Universal Robots PolyScope program: Test Script Calcs.urp

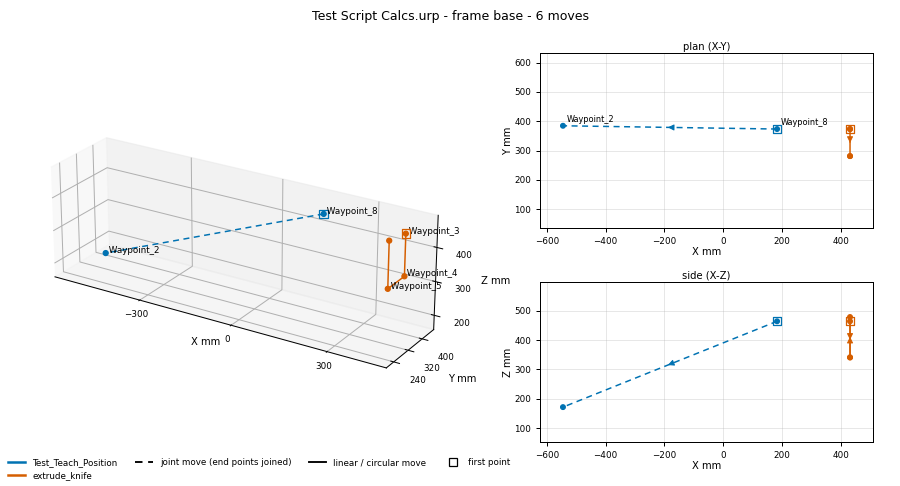
[picture p0: tool path of Test Script Calcs.urp in frame base, 6 of 9 moves have a stored position in this frame; points joined in program order, loops and branches not executed]
Program Test Script Calcs (installation=default directory=/programs createdIn=5.14.5 lastSavedIn=5.14.5 robotSerialNumber=20236801216)
Calibrated DH parameters: a=[-0.000021, -0.748897, -0.28186, -0.00004, -0.000055, 0]; d=[0.236225, -424.082933, -1564.66872, 1988.95162, 0.159094, 0.153873]; alpha=[1.570844, 0.001002, 0.000337, 1.571488, -1.569996, 0]; deltaTheta=[0, -0.516316, 5.626292, 1.173211, 0.000001, 0]
InitVariablesNode variables(variable(name=freedrive_m_var, expression=False))
Robot Program (runOnlyOnce=true)
  Script: Test_Teach_Position()
  Script: Corner_Homing_BRB()
  Script: extrude_knife()
  Script: test_script_calcs2()
SubProgram Test_Teach_Position (keepSynchronizedWithDisk=false) programFile=/programs/Test Teach Position.urp
  SafeHome (positionOptionType=SPEED_AND_ACCELERATION speed=1.047198 acceleration=1.396263 nextMotionTime=2)
  MoveL speed 250 mm/s, acceleration 1200 mm/s^2 (useActiveTCP=true) feature=Base
    Waypoint Waypoint_8: TCP in base x=183.613 y=373.491 z=464.002 mm, rx=0 ry=3.1416 rz=0 rad; joints [-144.817, -120.486, 148.461, -117.931, -90.033, 125.101] deg; TCP offset x=0 y=0 z=19 mm, rx=0 ry=0 rz=0 rad
    'move welder up out of holder'
  MoveJ speed 60 deg/s, acceleration 80 deg/s^2 (useActiveTCP=true) feature=Base
    Waypoint Waypoint_2: TCP in base x=-545.552 y=384.638 z=171.639 mm, rx=0.6685 ry=-1.9493 rz=1.7266 rad; joints [-60.534, -62.274, 125.356, -70.677, -59.999, 145.088] deg
  freedrive_m_var := False
  freedrive_m_var := True
  Popup Message (haltProgram=false message=Move the robot to the peg center, then click 'Continue' inputType=Text)
  freedrive_m_var := False
  Wait Sleep waitTime=0.25
  Script: sync()
  tcp_pose := get_actual_joint_positions()
SubProgram Corner_Homing_BRB (keepSynchronizedWithDisk=false) programFile=/programs/Corner Homing BRB.urp
  'Use this program when tool is already positioned close to corner (back right bottom corner)'
  'tool flange will seek all 3 sides and then bring tcp to the corner'
  Script: align_tcp_left()
  'right side'
  MoveL speed 250 mm/s, acceleration 1200 mm/s^2 (useActiveTCP=true) feature=Base
    MoveDirectionNode (selectedDirection=XMinus)
      Until DISTANCE (allowActions=false deceleration=3 distanceNodeType=STOP) Distance=0.05; motionParameters(blendRadius=0)
  MoveL speed 50 mm/s, acceleration 1200 mm/s^2 (useActiveTCP=true) feature=Base
    MoveDirectionNode (selectedDirection=YMinus)
      Until TOOL_CONTACT_DETECTION (allowActions=false retraction=0 decelerationAcceleration=3 decelerationAngularAcceleration=34.906585)
  p11 := get_actual_tcp_pose()
  MoveL speed 250 mm/s, acceleration 1200 mm/s^2 (useActiveTCP=true) feature=Base
    MoveDirectionNode (selectedDirection=YPlus)
      Until DISTANCE (allowActions=false deceleration=3 distanceNodeType=STOP) Distance=0.05; motionParameters(blendRadius=0)
  MoveL speed 250 mm/s, acceleration 1200 mm/s^2 (useActiveTCP=true) feature=Base
    MoveDirectionNode (selectedDirection=XMinus)
      Until DISTANCE (allowActions=false deceleration=3 distanceNodeType=STOP) Distance=0.05; motionParameters(blendRadius=0)
  MoveL speed 50 mm/s, acceleration 1200 mm/s^2 (useActiveTCP=true) feature=Base
    MoveDirectionNode (selectedDirection=YMinus)
      Until TOOL_CONTACT_DETECTION (allowActions=false retraction=0 decelerationAcceleration=3 decelerationAngularAcceleration=34.906585)
  p12 := get_actual_tcp_pose()
  MoveL speed 250 mm/s, acceleration 1200 mm/s^2 (useActiveTCP=true) feature=Base
    MoveDirectionNode (selectedDirection=YPlus)
      Until DISTANCE (allowActions=false deceleration=3 distanceNodeType=STOP) Distance=0.05; motionParameters(blendRadius=0)
  MoveL speed 250 mm/s, acceleration 1200 mm/s^2 (useActiveTCP=true) feature=Base
    MoveDirectionNode (selectedDirection=XPlus)
      Until DISTANCE (allowActions=false deceleration=3 distanceNodeType=STOP) Distance=0.2; motionParameters(blendRadius=0)
  Script: align_tcp_forward()
  'back side'
  MoveL speed 250 mm/s, acceleration 1200 mm/s^2 (useActiveTCP=true) feature=Base
    MoveDirectionNode (selectedDirection=YMinus)
      Until DISTANCE (allowActions=false deceleration=3 distanceNodeType=STOP) Distance=0.1; motionParameters(blendRadius=0)
  MoveL speed 50 mm/s, acceleration 1200 mm/s^2 (useActiveTCP=true) feature=Base
    MoveDirectionNode (selectedDirection=XMinus)
      Until TOOL_CONTACT_DETECTION (allowActions=false retraction=0 decelerationAcceleration=3 decelerationAngularAcceleration=34.906585)
  p21 := get_actual_tcp_pose()
  MoveL speed 250 mm/s, acceleration 1200 mm/s^2 (useActiveTCP=true) feature=Base
    MoveDirectionNode (selectedDirection=XPlus)
      Until DISTANCE (allowActions=false deceleration=3 distanceNodeType=STOP) Distance=0.05; motionParameters(blendRadius=0)
  MoveL speed 250 mm/s, acceleration 1200 mm/s^2 (useActiveTCP=true) feature=Base
    MoveDirectionNode (selectedDirection=YMinus)
      Until DISTANCE (allowActions=false deceleration=3 distanceNodeType=STOP) Distance=0.05; motionParameters(blendRadius=0)
  MoveL speed 50 mm/s, acceleration 1200 mm/s^2 (useActiveTCP=true) feature=Base
    MoveDirectionNode (selectedDirection=XMinus)
      Until TOOL_CONTACT_DETECTION (allowActions=false retraction=0 decelerationAcceleration=3 decelerationAngularAcceleration=34.906585)
  p22 := get_actual_tcp_pose()
  MoveL speed 250 mm/s, acceleration 1200 mm/s^2 (useActiveTCP=true) feature=Base
    MoveDirectionNode (selectedDirection=XPlus)
      Until DISTANCE (allowActions=false deceleration=3 distanceNodeType=STOP) Distance=0.05; motionParameters(blendRadius=0)
  'regroup for up turn'
  MoveL speed 250 mm/s, acceleration 1200 mm/s^2 (useActiveTCP=true) feature=Base
    MoveDirectionNode (selectedDirection=XPlus)
      Until DISTANCE (allowActions=false deceleration=3 distanceNodeType=STOP) Distance=0.2; motionParameters(blendRadius=0)
    MoveDirectionNode (selectedDirection=YPlus)
      Until DISTANCE (allowActions=false deceleration=3 distanceNodeType=STOP) Distance=0.4; motionParameters(blendRadius=0)
  MoveL speed 250 mm/s, acceleration 1200 mm/s^2 (useActiveTCP=true) feature=Base
    MoveDirectionNode (selectedDirection=ZMinus)
      Until DISTANCE (allowActions=false deceleration=3 distanceNodeType=STOP) Distance=0.1; motionParameters(blendRadius=0)
  Script: align_tcp_up()
  MoveL speed 250 mm/s, acceleration 1200 mm/s^2 (useActiveTCP=true) feature=Base
    MoveDirectionNode (selectedDirection=XMinus)
      Until DISTANCE (allowActions=false deceleration=3 distanceNodeType=STOP) Distance=0.25; motionParameters(blendRadius=0)
    MoveDirectionNode (selectedDirection=YMinus)
      Until DISTANCE (allowActions=false deceleration=3 distanceNodeType=STOP) Distance=0.3; motionParameters(blendRadius=0)
  'bottom side'
  MoveL speed 250 mm/s, acceleration 1200 mm/s^2 (useActiveTCP=true) feature=Base
    MoveDirectionNode (selectedDirection=YMinus)
      Until DISTANCE (allowActions=false deceleration=3 distanceNodeType=STOP) Distance=0.12; motionParameters(blendRadius=0)
  MoveL speed 50 mm/s, acceleration 1200 mm/s^2 (useActiveTCP=true) feature=Base
    MoveDirectionNode (selectedDirection=ZPlus)
      Until TOOL_CONTACT_DETECTION (allowActions=false retraction=0 decelerationAcceleration=3 decelerationAngularAcceleration=34.906585)
  p3 := get_actual_tcp_pose()
  MoveL speed 250 mm/s, acceleration 1200 mm/s^2 (useActiveTCP=true) feature=Base
    MoveDirectionNode (selectedDirection=ZMinus)
      Until DISTANCE (allowActions=false deceleration=3 distanceNodeType=STOP) Distance=0.05; motionParameters(blendRadius=0)
  MoveL speed 250 mm/s, acceleration 1200 mm/s^2 (useActiveTCP=true) feature=Base
    MoveDirectionNode (selectedDirection=XPlus)
      Until DISTANCE (allowActions=false deceleration=3 distanceNodeType=STOP) Distance=0.1; motionParameters(blendRadius=0)
    MoveDirectionNode (selectedDirection=YPlus)
      Until DISTANCE (allowActions=false deceleration=3 distanceNodeType=STOP) Distance=0.1; motionParameters(blendRadius=0)
SubProgram extrude_knife (keepSynchronizedWithDisk=false) programFile=/programs/extrude_knife.urp
  'Move to bucket'
  MoveJ speed 60 deg/s, acceleration 80 deg/s^2 (useActiveTCP=true) feature=Base
    Waypoint Waypoint_3: TCP in base x=432.121 y=373.496 z=463.993 mm, rx=0 ry=-3.1416 rz=0 rad; joints [-159.589, -103.956, 140.658, -126.656, -90.019, 110.321] deg
  MoveL speed 250 mm/s, acceleration 1200 mm/s^2 (useActiveTCP=true) feature=Base
    Waypoint Waypoint_4: TCP in base x=432.138 y=373.502 z=340.884 mm, rx=0 ry=3.1416 rz=0 rad; joints [-159.596, -94.144, 147.137, -142.947, -90.01, 110.313] deg
  'extrude out a foot'
  Wait Sleep waitTime=6
  MoveL speed 40 mm/s, acceleration 1200 mm/s^2 (useActiveTCP=true) feature=Base
    'slice over knife'
    Waypoint Waypoint_5: TCP in base x=432.16 y=281.352 z=340.893 mm, rx=0 ry=3.1416 rz=0 rad; joints [-169.69, -98.838, 150.801, -141.919, -90.013, 100.22] deg
  MoveL speed 250 mm/s, acceleration 1200 mm/s^2 (useActiveTCP=true) feature=Base
    Waypoint Waypoint_6: TCP in base x=432.128 y=281.346 z=478.493 mm, rx=0 ry=-3.1416 rz=0 rad; joints [-169.679, -110.118, 142.836, -122.671, -90.025, 100.232] deg
    'raise up away from knife'
SubProgram test_script_calcs2 (keepSynchronizedWithDisk=false) programFile=/programs/test_script_calcs2.urp
  point1 := get_actual_tcp_pose()
  point2 := get_actual_tcp_pose()
  point3 := get_actual_tcp_pose()
  point4 := get_actual_tcp_pose()
  Script file /programs/analyze_touchpoints.script
    | # comment get the z
    | zcoord=p3[2]
    | 
    | # get the raw points from the first line
    | l1p1x=p11[0]
    | l1p1y=p11[1]
    | l1p2x=p12[0]
    | l1p2y=p12[1]
    | 
    | # equate the first line in 2d space
    | ml1 = (l1p2y-l1p1y) / (l1p2x-l1p1x)
    | 
    | # b = y - mx
    | bl1 = l1p1y - ml1 * l1p1x
    | 
    | # get the raw points from the second line
    | l2p1x=p21[0]
    | l2p1y=p21[1]
    | l2p2x=p22[0]
    | l2p2y=p22[1]
    | 
    | # equate the second line in 2d space
    | ml2 = (l2p2y-l2p1y) / (l2p2x-l2p1x)
    | 
    | # b = y - mx
    | bl2 = l2p1y - ml2 * l2p1x
    | 
    | 
    | # find the intersection of the two lines
    | # m1x+b1 = m2x+b2
    | # m1x - m2x = b2 - b1
    | # x = (b2-b1) / (m1-m2)
    | xintersect = (bl2-bl1) / (ml1-ml2)
    | yintersect = ml1 * xintersect + bl1
    | 
    | 
    | # find locations 8 inches away from  intersect point
    | # CONST
    | welddistance = 8
    | roundoverdistance = .25
    | zup = .375
    | # inches
    | wd = welddistance * 25.4 / 1000
    | rod = roundoverdistance * 25.4 / 1000
    | zup = zup * 25.4 / 1000
    | 
    | #define a vector from the intersection to the second point on the first line
    | l1delxfull = l1p2x - xintersect
    | l1delyfull = l1p2y - yintersect
    | 
    | l1delmag = sqrt(l1delxfull*l1delxfull + l1delyfull*l1delyfull)
    | 
    | l1delxunit = l1delxfull / l1delmag
    | l1delyunit = l1delyfull / l1delmag
    | 
    | # now we have the unit vector. extend the weld distance from the intersection
    | x = xintersect + l1delxunit * wd
    | y = yintersect + l1delyunit * wd
    | z = zcoord + zup
    | 
    | point1 = p[x,y,z,1.570796,0,0] # dummy orientation for now
    | 
    | x = xintersect + l1delxunit * rod
    | y = yintersect + l1delyunit * rod
    | 
    | point2 = p[x,y,z,1.570796,0,0]
    | 
    | #define a vector from the intersection to the second point on the second line
    | l2delxfull = l2p2x - xintersect
    | l2delyfull = l2p2y - yintersect
    | 
    | l2delmag = sqrt(l2delxfull*l2delxfull + l2delyfull*l2delyfull)
    | 
    | l2delxunit = l2delxfull / l2delmag
    | l2delyunit = l2delyfull / l2delmag
    | 
    | # now we have the unit vector. extend the weld distance from the intersection
    | x = xintersect + l2delxunit * wd
    | y = yintersect + l2delyunit * wd
    | 
    | point4 = p[x,y,z,0,-1.570796,0]
    | 
    | x = xintersect + l2delxunit * rod
    | y = yintersect + l2delyunit * rod
    | 
    | point3 = p[x,y,z,0,-1.570796,0]
    | 
    | pointintersect = p[xintersect,yintersect,zcoord,1.570796,0,0]
    | pointapproach1 = p[xintersect+0.1,yintersect+0.1,z,1.570796,0,0]
    | pointapproach2 = p[point1[0] + 0.1, point1[1], point1[2], point1[3], point1[4], point1[5]]
    | 
    | 
    | # the orthogonal direction 1 IS the vector direction 2 (and vice versa)
    | 
    | # but for now, just use orthogonal angles
  Script file /programs/move_weld_brb.script
    | # this script actually moves the robot along the path
    | # for testing. no welder attached, no orientation decided
    | 
    | movej(pointapproach1, a=1.2, v=0.25)
    | 
    | movel(pointapproach2, a=1.2, v=0.25)
    | 
    | movel(point1, a=1.2, v=0.25)
    | 
    | movel(point2, a=1.2, v=0.25)
    | 
    | movel(point3, a=1.2, v=0.25)
    | 
    | movel(point4, a=1.2, v=0.25)
    | 
    | movel(pointapproach1, a=1.2, v=0.25)
SubProgram align_tcp_left (keepSynchronizedWithDisk=false) programFile=/programs/align_tcp_left.urp
  'this program aligns the tcp parallel to the y direction'
  cp := get_actual_tcp_pose()
  aligned_y_pose := p[cp[0],cp[1],cp[2],1.570796,0,0]
  MoveJ speed 60 deg/s, acceleration 80 deg/s^2 (useActiveTCP=true) feature=Base
    Waypoint Variable (Variable): variable(name=aligned_y_pose)
SubProgram align_tcp_up (keepSynchronizedWithDisk=false) programFile=/programs/align_tcp_up.urp
  'this program aligns the tcp parallel to the y direction'
  cp := get_actual_tcp_pose()
  aligned_y_pose := p[cp[0],cp[1],cp[2],0,0,0]
  MoveJ speed 60 deg/s, acceleration 80 deg/s^2 (useActiveTCP=true) feature=Base
    Waypoint Variable (Variable): variable=aligned_y_pose
SubProgram align_tcp_forward (keepSynchronizedWithDisk=false) programFile=/programs/align_tcp_forward.urp
  'this program aligns the tcp parallel to the y direction'
  cp := get_actual_tcp_pose()
  aligned_y_pose := p[cp[0],cp[1],cp[2],0,-1.570796,0]
  MoveJ speed 60 deg/s, acceleration 80 deg/s^2 (useActiveTCP=true) feature=Base
    Waypoint Variable (Variable): variable=aligned_y_pose
Thread Thread_1 (runOnlyOnce=false)
  Loop While (checkContinuously=false) expression=True
    If freedrive_m_var≟ True
      Script: freedrive_mode()
    Else 
      Script: end_freedrive_mode()
    Script: sync()
